FUNCTION_BLOCK FB_PullWheel EXTENDS FB_PackML_BaseModule
VAR
    // Sub module definitions here

    // List of sub modules
    ipSubModules_Init : ARRAY[1..Parameters_PackML_Base.MAX_NO_OF_SUBMODULES] OF I_PackML_BaseModule := [];

    // Component definitions here
    LeftPullWheel     : FB_Component_BasicSlaveAxis := (Name := 'Left');
    RightPullWheel    : FB_Component_BasicSlaveAxis := (Name := 'Right');
    PullWheelCylinder : FB_Cylinder                 := (Name := 'Cylinder');

    // List of Components
    ipComponents_Init : ARRAY[1..Parameters_PackML_Base.MAX_NO_OF_COMPONENTS] OF I_ComponentBase
        := [LeftPullWheel, RightPullWheel, PullWheelCylinder];

    //Alarms for this module
    PullWheelAlarms : ARRAY[1..PULL_WHEELS_ALARM_COUNT] OF FB_TcAlarm;

	//Data for recipe
	Recipe : ST_PullWheelsRecipe;
    (*Parameters from PackTags for module
    _Param  : ARRAY[1..10] OF ST_Descriptor2;*)
    _Report : ARRAY[1..10] OF ST_Descriptor2;

    //HMI Control for EM
    fbControlSourceHMI : FB_ControlSource_HMI;
END_VAR

VAR CONSTANT

    //reports 
    FAULT : INT := 1;

    //Alarms
    PULL_WHEELS_ALARM_COUNT : INT := 5;
END_VAR

//Simulation variables for messaging
VAR
    ErrorInput : BOOL;
    WarnInput  : BOOL;
    InfoInput  : BOOL;
END_VAR

METHOD PROTECTED Aborting
VAR_INPUT
END_VAR
CASE SequenceState OF
    0:
        NoStateTasksToComplete := FALSE;
        SequenceState          := SequenceState + 10;
    10:
        LeftPullWheel.Stop();
        RightPullWheel.Stop();
        IF LeftPullWheel.Stopped AND RightPullWheel.Stopped THEN
            SequenceState := SequenceState + 10;
        END_IF
    20:
        // Disable here
        LeftPullWheel.Disable();
        RightPullWheel.Disable();
        PullWheelCylinder.Retract();

        // Check not enabled here
        IF NOT LeftPullWheel.Enabled AND NOT RightPullWheel.Enabled AND PullWheelCylinder.Retracted THEN
            SequenceState := SequenceState + 10;
        END_IF

        StateTasksComplete := TRUE;
END_CASE

SUPER^.Aborting();
END_METHOD

PROPERTY Acceleration : LREAL
SET
Recipe.LeftAxis.Acceleration := Acceleration;
Recipe.RightAxis.Acceleration := Acceleration;
END_SET
END_PROPERTY

METHOD PROTECTED Clearing
VAR_INPUT
END_VAR
CASE SequenceState OF
    0:
        NoStateTasksToComplete := FALSE;
        SequenceState          := SequenceState + 10;
    10:
        //Reset any alarms that get latched
        PullWheelAlarms[E_PullWheels.StartTimeout].Clear(0, 0);
        SequenceState := SequenceState + 10;
    20:
        // Enable here
        LeftPullWheel.Enable();
        RightPullWheel.Enable();

        // Check enabled here
        IF LeftPullWheel.Enabled AND RightPullWheel.Enabled THEN
            SequenceState := SequenceState + 10;
        END_IF
    30:
        StateTasksComplete := TRUE;
END_CASE

SUPER^.Clearing();
END_METHOD

METHOD PROTECTED CreateEvents
VAR_INPUT
END_VAR
// Add your event creation here
F_CreateAllEventsInClass(Alarms     := PullWheelAlarms,
                         ClassSize  := SIZEOF(TC_EVENTS.PullWheels),
                         pInitEvent := ADR(TC_EVENTS.PullWheels.InitReferenceEvent),
                         Prefix     := _Name);

// Super call to base
SUPER^.CreateEvents();
END_METHOD

METHOD CyclicLogic
VAR_INPUT
END_VAR
IF NOT _InitComplete THEN
    _InitComplete := Initialize();
    RETURN;
END_IF

SUPER^.CyclicLogic();

//HMI control for EM
fbControlSourceHMI.CyclicLogic();

//Set the current alarm severity for this module
_CurrentAlarmSeverity := F_GetMaxSeverityRaised(Alarms := PullWheelAlarms, CurrentSeverity := _CurrentAlarmSeverity);

//Simulate Alarm Messaging
CyclicLogic_Simulation();
END_METHOD

METHOD CyclicLogic_Simulation
VAR_INPUT
END_VAR

VAR_INST
END_VAR
(*	
This is just for testing. Real hardware can be setup in other places
Here the alarms will raise and clear on its own if the input changes	
*)

//Generic Alarms for Testing
IF ErrorInput AND NOT PullWheelAlarms[E_PullWheels.AlarmMessage].bRaised THEN
    RaiseAlarm2Args(PullWheelAlarms[E_PullWheels.AlarmMessage], '', '');
ELSIF NOT ErrorInput AND PullWheelAlarms[E_PullWheels.AlarmMessage].bRaised THEN
    PullWheelAlarms[E_PullWheels.AlarmMessage].Clear(0, 0);
END_IF

IF WarnInput AND NOT PullWheelAlarms[E_PullWheels.WarnMessage].bRaised THEN
    RaiseAlarm2Args(PullWheelAlarms[E_PullWheels.WarnMessage], '', '');
ELSIF NOT WarnInput AND PullWheelAlarms[E_PullWheels.WarnMessage].bRaised THEN
    PullWheelAlarms[E_PullWheels.WarnMessage].Clear(0, 0);
END_IF

IF InfoInput AND NOT PullWheelAlarms[E_PullWheels.InfoMessage].bRaised THEN
    RaiseAlarm2Args(PullWheelAlarms[E_PullWheels.InfoMessage], '', '');
ELSIF NOT InfoInput AND PullWheelAlarms[E_PullWheels.InfoMessage].bRaised THEN
    PullWheelAlarms[E_PullWheels.InfoMessage].Clear(0, 0);
END_IF
END_METHOD

METHOD PROTECTED Execute
VAR_INPUT
END_VAR
// Function based on mode.  NO need to make SUPER^.Executing() since it does nothing.
CASE _CurrentMode OF
    E_PMLUnitMode.ePMLUnitMode_Production:
        IF LeftPullWheel.InPosition AND NOT LeftPullWheel.Busy THEN
            PullWheelCylinder.Retract();
            IF PullWheelCylinder.Retracted THEN
                StateComplete();
            END_IF
        END_IF
    E_PMLUnitMode.ePMLUnitMode_Maintenance:
        ;
    E_PMLUnitMode.ePMLUnitMode_Manual:
        ;
END_CASE
END_METHOD

//! @summary Basic module initialization logic
METHOD PROTECTED Initialize : BOOL;
VAR
    i                        : UDINT;
    varInfo                  : __SYSTEM.VAR_INFO;
    AllSubUnitsInitialized   : BOOL := TRUE;
    AllComponentsInitialized : BOOL := TRUE;
END_VAR

//! @description This method is called by <c>CyclicLogic()</c> as required
Initialize := FALSE;
CASE DescendantSequenceState OF
    0:
        // Define the interfaces to the different subunits (Must take place before SUPER^.initialize call)
        FOR i := 1 TO SPT_BaseTypes.Parameters_PackML_Base.MAX_NO_OF_SUBMODULES DO
            ipSubModules[i] := ipSubModules_Init[i];
        END_FOR

        FOR i := 1 TO SPT_BaseTypes.Parameters_PackML_Base.MAX_NO_OF_COMPONENTS DO
            ipComponents[i] := ipComponents_Init[i];
        END_FOR

        _LogModeChanges         := FALSE;
        _LogStateChanges        := FALSE;
        DescendantSequenceState := DescendantSequenceState + 10;
    10:
        //Setup Custom modes here

        (*CustomModes(eMode                          :=,
                    sName                          :=,
                    bDisableClearing               :=,
                    bDisableStarting               :=,
                    bDisableSuspended              :=,
                    bDisableStopping               :=,
                    bDisableAborting               :=,
                    bDisableHolding                :=,
                    bDisableHeld                   :=,
                    bDisableUnholding              :=,
                    bDisableSuspending             :=,
                    bDisableUnsuspending           :=,
                    bDisableResetting              :=,
                    bDisableIdle                   :=,
                    bDisableCompleting             :=,
                    bDisableComplete               :=,
                    bEnableUnitModeChangeStopped   :=,
                    bEnableUnitModeChangeIdle      :=,
                    bEnableUnitModeChangeSuspended :=,
                    bEnableUnitModeChangeExecute   :=,
                    bEnableUnitModeChangeAborted   :=,
                    bEnableUnitModeChangeHeld      :=,
                    bEnableUnitModeChangeComplete  :=,
                    bError                         =>,
                    nErrorId                       =>);*)
        DescendantSequenceState := DescendantSequenceState + 10;
    20:
        //Copy Mode names
        FOR i := 1 TO 3 DO
            ModeNames[i] := F_UnitModeToString(UDINT_TO_DINT(i));
        END_FOR

        Initialize_TagData();
		RegisterExternalController(Controller := fbControlSourceHMI);
		fbControlSourceHMI.CyclicLogic();
        DescendantSequenceState := DescendantSequenceState + 10;
    30:
        //Call the Super
        IF SUPER^.Initialize() THEN
            DescendantSequenceState := DescendantSequenceState + 10;
        END_IF
    40:
        Initialize := TRUE;
END_CASE
END_METHOD

METHOD Initialize_TagData
VAR_INPUT
END_VAR
// Reports
_Report[FAULT].ID    := TO_DINT(1 * 10 + 1);
_Report[FAULT].Name  := 'Fault ID';
_Report[FAULT].Unit  := 'n/a';

//Recipe
Recipe.Length := 100;
Recipe.LeftAxis.Velocity := 100;
Recipe.LeftAxis.Acceleration := 1000;
Recipe.RightAxis.Velocity := 100;
Recipe.RightAxis.Acceleration := 1000;
END_METHOD

PROPERTY Length : LREAL
GET
Length := Recipe.Length;
END_GET
SET
Recipe.Length := Length;
END_SET
END_PROPERTY

METHOD RaiseAlarm2Args
VAR_IN_OUT
    Alarm : FB_TcAlarm; //Alarm to be raised
END_VAR

VAR_INPUT
    String_1 : STRING; //First String Parameter (The Name of this component will be applied first automatically)
    String_2 : STRING; //Second String Parameter
END_VAR
F_RaiseAlarmWithStringParameters(Alarm    := Alarm,
                                 String_1 := Name,
                                 String_2 := String_1,
                                 String_3 := String_2);
END_METHOD

METHOD PROTECTED Resetting
VAR_INPUT
END_VAR
CASE _CurrentMode OF
    //=================================PRODUCTION MODE==================================
    E_PMLUnitMode.ePMLUnitMode_Production:
        CASE SequenceState OF
            0:
                NoStateTasksToComplete := FALSE;
                SequenceState          := SequenceState + 10;
            10:
                /// No reason to gear to the master LeftPullWheel.Master1  REF= MAIN.ApicoSeed.Master.Axis;
                RightPullWheel.Master1 REF= LeftPullWheel.Axis;

                ///LeftPullWheel.GearIn();
                RightPullWheel.GearIn();
                SequenceState := SequenceState + 10;
            20:
                IF (*LeftPullWheel.InGear AND*) RightPullWheel.InGear THEN
                    StateTasksComplete := TRUE;
                END_IF
        END_CASE

    //=================================MAINTENANCE & MANUAL MODE==================================	
    E_PMLUnitMode.ePMLUnitMode_Maintenance, E_PMLUnitMode.ePMLUnitMode_Manual:
        ;
END_CASE

SUPER^.Resetting();
END_METHOD

METHOD PROTECTED Starting
VAR_INPUT
END_VAR

VAR_INST
    StartTimer : TON;
END_VAR
CASE _CurrentMode OF
    //=================================PRODUCTION MODE==================================
    E_PMLUnitMode.ePMLUnitMode_Production:
        CASE SequenceState OF
            0:
                // Delay 1 scan to make sure timer is off.  Not guarnteed from last time where it finished.
                NoStateTasksToComplete := FALSE;
                SequenceState          := SequenceState + 10;
            10:
                PullWheelCylinder.Extend();
                IF PullWheelCylinder.Extended THEN
                    NoStateTasksToComplete     := FALSE;
                    LeftPullWheel.Velocity     := Recipe.LeftAxis.Velocity;
                    LeftPullWheel.Acceleration := Recipe.LeftAxis.Acceleration;
                    LeftPullWheel.MoveRelative(Distance := Recipe.Length, FALSE);
                    SequenceState := SequenceState + 10;
                END_IF
            20:
                IF LeftPullWheel.Busy THEN
                    SequenceState := SequenceState + 10;
                END_IF

                IF StartTimer.Q AND NOT PullWheelAlarms[E_PullWheels.StartTimeout].bRaised THEN
                    RaiseAlarm2Args(PullWheelAlarms[E_PullWheels.StartTimeout], '', '');
                    SequenceState := SequenceState + 10;
                END_IF
            30:
                StateTasksComplete := TRUE;
        END_CASE

    //=================================MAINTENANCE & MANUAL MODE==================================
    E_PMLUnitMode.ePMLUnitMode_Maintenance, E_PMLUnitMode.ePMLUnitMode_Manual:
        ;
END_CASE

SUPER^.Starting();
StartTimer(IN := ((SequenceState = 10) OR (SequenceState = 20)), PT := T#3S);
END_METHOD

METHOD PROTECTED Stopping
VAR_INPUT
END_VAR
CASE _CurrentMode OF
    //=================================PRODUCTION MODE==================================
    E_PMLUnitMode.ePMLUnitMode_Production:
        CASE SequenceState OF
            0:
                NoStateTasksToComplete := FALSE;
                PullWheelCylinder.Retract();
                SequenceState := SequenceState + 10;
            10:
                IF PullWheelCylinder.Retracted THEN
                    SequenceState := SequenceState + 10;
                END_IF
            20:
                StateTasksComplete := TRUE;
        END_CASE

    //=================================MAINTENANCE & MANUAL MODE==================================
    E_PMLUnitMode.ePMLUnitMode_Maintenance, E_PMLUnitMode.ePMLUnitMode_Manual:
        ;
END_CASE

SUPER^.Stopping();
END_METHOD

PROPERTY Velocity : LREAL
SET
Recipe.LeftAxis.Velocity := Velocity;
Recipe.RightAxis.Velocity := Velocity;
END_SET
END_PROPERTY

END_FUNCTION_BLOCK

(* stored: Version 1.1.0.1, ProductVersion 3.1.4024.12
   POU FB_PullWheel: Id {496b17f1-4b0a-4954-89f4-eec9ef72b2f5}, SpecialFunc None
   Folder I_CyclicFB: Id {1cfc12b1-3488-4708-a9c0-7f5e3200922e}
   Folder Methods: Id {7ea91248-a559-47e3-a56f-a225596d5ea4}
   Folder Acting States: Id {30d294a1-5cf9-40fa-a3c4-3abcbefdbe05}
   Folder Waiting States: Id {ce7f79c0-77aa-4f06-a5c0-97eff08c325c}
   Folder Properties: Id {d979cebd-5da6-4378-800d-7adb88acdfab}
   Method Aborting: Id {4c3de770-a28d-4000-93d6-e12df93294dd}
   Property Acceleration: Id {fb737272-8121-443f-bb81-17cc6deb00e3}
   Set Set: Id {a82221d7-d213-426a-9fb3-1813ff8529dc}
   Method Clearing: Id {0331837f-22a2-46ed-b836-140316680a45}
   Method CreateEvents: Id {4ec0ace2-c308-44b2-84a1-60ba649bd547}
   Method CyclicLogic: Id {02def406-fced-425b-89cd-43b7d8052b02}
   Method CyclicLogic_Simulation: Id {848790f4-6965-4320-b33a-fb32f7f918da}
   Method Execute: Id {24f2a84a-cfe1-4269-89c3-0ab58d2e748b}
   Method Initialize: Id {b4a0fd62-4385-4420-ae43-9bea35a3f798}
   Method Initialize_TagData: Id {32a2e019-abce-425f-8e3c-cc5fca6b6f69}
   Property Length: Id {25f83960-2850-4c98-aac0-0474e792dc9b}
   Get Get: Id {49a64ec1-b283-4c39-b495-d337d077c39a}
   Set Set: Id {62003e52-0dea-4a17-a8a3-a51e509c6ad2}
   Method RaiseAlarm2Args: Id {3b444795-a02f-4331-ab15-8dec5e002fb2}
   Method Resetting: Id {c85d70ed-952c-4c53-9986-231b7ace540a}
   Method Starting: Id {c8ce40ea-dea4-41f3-bfcc-e10ad34fff3f}
   Method Stopping: Id {7d6ebde9-664e-4d12-ba2e-b6039c72785e}
   Property Velocity: Id {95139607-01c7-400b-9b34-9fbd90d24f62}
   Set Set: Id {e26bea52-2635-4098-a40e-4dd141afac28} *)
